INTERFACE I_Station_LinkedList

METHOD AddHeadValue : ST_STATION_LIST_RESULT
VAR_INPUT
  stData        : ST_STATION_MOVER_DATA;
END_VAR
END_METHOD

METHOD AddTailValue : ST_STATION_LIST_RESULT
VAR_INPUT
  stData          : ST_STATION_MOVER_DATA;
END_VAR
END_METHOD

PROPERTY Count : UDINT
GET
END_GET
END_PROPERTY

PROPERTY Data : ARRAY[0..MAX_LIST_NODES] OF ST_STATION_MOVER_DATA
GET
END_GET
END_PROPERTY

PROPERTY Free : UDINT
GET
END_GET
END_PROPERTY

METHOD GetHead : ST_STATION_LIST_RESULT
VAR_INPUT
END_VAR
END_METHOD

METHOD InitList : BOOL
END_METHOD

PROPERTY Nodes : ARRAY[0..MAX_LIST_NODES] OF T_LinkedListEntry
GET
END_GET
END_PROPERTY

METHOD RemoveHeadValue : ST_STATION_LIST_RESULT
VAR_INPUT
END_VAR
END_METHOD

END_INTERFACE

(* stored: Version 1.1.0.1, ProductVersion 3.1.4024.12
   Itf I_Station_LinkedList: Id {bba57127-e721-4bbe-8c2d-84a6c8a5d1d5}
   Method AddHeadValue: Id {e8a70d07-6516-42f6-93c7-859646a5c0dc}
   Method AddTailValue: Id {9395ab5b-196d-467d-bd28-d48760300fd3}
   Property Count: Id {ef13f797-d18d-44e3-b2f2-078b68470a66}
   Get Get: Id {56dc153c-c249-4b39-ab81-2c89b2509f9d}
   Property Data: Id {4916ec1b-ea75-477a-96cf-c9fddd620d7d}
   Get Get: Id {07fb5d63-ce41-4eed-8049-5f2619f2dbbc}
   Property Free: Id {3bd7968f-150b-4166-97a5-4f3940afb6d8}
   Get Get: Id {98bcd5d7-2205-47a6-a663-44a5cf6fd037}
   Method GetHead: Id {3a7c5f05-4248-4b04-9fce-2e4b6672aa14}
   Method InitList: Id {1e78bd58-b1da-4b47-b6ac-b628533e03b9}
   Property Nodes: Id {76f63815-da22-4ca9-b984-7bf187be2355}
   Get Get: Id {2f494f6f-2776-4027-8735-68b6c0532337}
   Method RemoveHeadValue: Id {f4b43985-8939-4777-b224-9ae48834d8bd} *)
